(* IEC 61131-3 sources: OpenPLCLogic/, 1 file *)

(* ---- FB_PumpControl.st ---- *)
FUNCTION_BLOCK FB_PumpControl
VAR_INPUT
    // Inputs
    StartManual : BOOL := FALSE;            // Manual start signal
    StopManual : BOOL := FALSE;             // Manual stop signal
    StartAuto : BOOL := FALSE;              // Automatic start signal
    StopAuto : BOOL := FALSE;               // Automatic stop signal
    SafetyInterlock : BOOL := TRUE;         // Safety interlock active (prevents operation)
    Pump1Running : BOOL := FALSE;           // Status of Pump 1
    Pump2Running : BOOL := FALSE;           // Status of Pump 2
    Pressure : REAL := 0.0;                 // Pump pressure
    BrakeCommand : BOOL := FALSE;           // Brake control command
    PriorityChangeTime : REAL := 1200.0;    // Time threshold (in seconds) after which priority changes
END_VAR
VAR_OUTPUT
    // Outputs
    Pump1Status : BOOL := FALSE;            // Pump 1 running status
    Pump2Status : BOOL := FALSE;            // Pump 2 running status
    BrakeStatus : BOOL := FALSE;            // Brake status (on/off)
    FaultStatus : BOOL := FALSE;            // Fault status (if any)
    PumpStatus : INT := 0;                  // Pump operational status (0=Off, 1=Running, 2=Fault)
END_VAR
VAR
    // Internal Variables
    PumpMode : INT := 0;                    // 0 = Manual, 1 = Auto
    PumpState : INT := 0;                   // 0 = Off, 1 = Running, 2 = Fault
    BrakeState : BOOL := FALSE;             // Brake applied or not
    Pump1Priority : BOOL := TRUE;           // Flag for load sharing (Pump 1 priority)
    TimeElapsed : REAL := 0.0;              // Time elapsed (in seconds)
    Pump1Load : REAL := 0.0;                // Load/pressure on Pump 1
    Pump2Load : REAL := 0.0;                // Load/pressure on Pump 2
    MaxLoad : REAL := 100.0;                // Max load threshold to avoid overload
    MaxPressure : REAL := 100.0;            // Maximum pressure limit (adjust as needed)
    Pump1Pressure : REAL := 0.0;            // Pressure for Pump 1
    Pump2Pressure : REAL := 0.0;            // Pressure for Pump 2
END_VAR

// Main Control Logic

    // Handle Safety Interlock - If interlock is active, stop the pumps
    IF NOT SafetyInterlock THEN
        FaultStatus := TRUE;
        PumpStatus := 2;  // Fault status
        Pump1Status := FALSE;
        Pump2Status := FALSE;
        BrakeStatus := TRUE; // Apply brake in case of interlock
        RETURN;
    END_IF

    // Handle Pump Operation Mode (Manual/Auto)
    IF PumpMode = 0 THEN  // Manual Mode
        // Manual Start/Stop Logic
        IF StartManual THEN
            // If not already running, start the pump
            IF NOT Pump1Running AND NOT Pump2Running THEN
                IF Pump1Priority THEN
                    Pump1Running := TRUE;
                ELSE
                    Pump2Running := TRUE;
                END_IF;
                PumpStatus := 1;  // Running
            END_IF;
        ELSIF StopManual THEN
            // Stop both pumps manually
            Pump1Running := FALSE;
            Pump2Running := FALSE;
            PumpStatus := 0;  // Stopped
        END_IF;
    ELSIF PumpMode = 1 THEN  // Automatic Mode
        // Automatically control pumps based on conditions (e.g., pressure or temperature)
        IF Pressure < 50.0 THEN  // If pressure is too low, start the pumps
            IF NOT Pump1Running AND NOT Pump2Running THEN
                IF Pump1Priority THEN
                    Pump1Running := TRUE;
                ELSE
                    Pump2Running := TRUE;
                END_IF;
                PumpStatus := 1;  // Running
            END_IF;
        ELSIF Pressure >= 50.0 THEN  // Stop pumps if pressure is sufficient
            Pump1Running := FALSE;
            Pump2Running := FALSE;
            PumpStatus := 0;  // Stopped
        END_IF;
    END_IF;

    // Manage Time-Based Pump Priority
    IF TimeElapsed >= PriorityChangeTime THEN
        Pump1Priority := NOT Pump1Priority;  // Change priority after the threshold time
        TimeElapsed := 0.0;  // Reset time counter
    END_IF;

    // Update pressure values for Pump1 and Pump2 based on system input
    Pump1Pressure := Pressure;  // Assume pressure input applies equally to both pumps (adjust as needed)
    Pump2Pressure := Pressure;  // Adjust this as per your system

    // Calculate load based on pressure
    Pump1Load := (Pump1Pressure / MaxPressure) * MaxLoad;
    Pump2Load := (Pump2Pressure / MaxPressure) * MaxLoad;

    // Handle Load Sharing (Tandem Operation)
    IF Pump1Running AND Pump2Running THEN
        // If both pumps are running, share load equally or adjust based on load
        IF Pump1Priority THEN
            // Check if Pump 1 is under heavy load based on pressure
            IF Pump1Load < MaxLoad THEN
                Pump2Running := FALSE;  // Stop Pump 2 to avoid overloading Pump 1
            END_IF;
        ELSE
            // Check if Pump 2 is under heavy load based on pressure
            IF Pump2Load < MaxLoad THEN
                Pump1Running := FALSE;  // Stop Pump 1 to avoid overloading Pump 2
            END_IF;
        END_IF;
    END_IF;

    // Update Pump Status
    IF Pump1Running THEN
        Pump1Status := TRUE;
    ELSE
        Pump1Status := FALSE;
    END_IF;

    IF Pump2Running THEN
        Pump2Status := TRUE;
    ELSE
        Pump2Status := FALSE;
    END_IF;

    // Handle Brake Control
    IF BrakeCommand THEN
        BrakeStatus := TRUE;  // Apply brake
        BrakeState := TRUE;   // Brake applied
    ELSE
        BrakeStatus := FALSE; // Release brake
        BrakeState := FALSE;  // Brake released
    END_IF;

    // Update Pump State
    IF NOT Pump1Running AND NOT Pump2Running THEN
        PumpState := 0;  // Pump is off
    ELSIF Pump1Running OR Pump2Running THEN
        PumpState := 1;  // Pump is running
    ELSE
        PumpState := 2;  // Fault state
    END_IF;
END_FUNCTION_BLOCK
